# B&R Automation Studio project CarWashSimu (part 2)

#### Main.st - Init, cyclic, exit code
```iecst
PROGRAM _INIT
	(* Insert code here *)

END_PROGRAM

PROGRAM _CYCLIC
	(* Insert code here *)
	HPAlarm;
	CASE sHPolishState OF
		enWAIT:
			IF iHPolish.Cmd.Start = TRUE THEN
				sHPolishState				:= enSTART;
			END_IF;
		enSTART:
			IF (iHPolish.IO.diSensHPolish1 = FALSE) AND (iHPolish.IO.diSensHPolish2 = FALSE) AND (iHPolish.IO.diSensHPolish3 = FALSE) AND (iHPolish.IO.diSensHPolish4 = FALSE) THEN
				iHPolish.IO.doRelayLower	:= TRUE;
				iHPolish.IO.doRelayLift		:= FALSE;
			END_IF;
			IF (iHPolish.IO.diSensHPolish1 = TRUE) AND (iHPolish.IO.diSensHPolish2 = FALSE) AND (iHPolish.IO.diSensHPolish3 = FALSE) AND (iHPolish.IO.diSensHPolish4 = FALSE) THEN
				iHPolish.IO.doRelayLower	:= FALSE;
				iHPolish.IO.doRelayLift		:= FALSE;
				iHPolish.IO.doRelayBrush	:= TRUE;
				sHPolishState				:= enOPERATION;
			END_IF;
		enOPERATION:
			IF (iHPolish.IO.diSensHPolish1 = TRUE) AND (iHPolish.IO.diSensHPolish2 = FALSE) AND (iHPolish.IO.diSensHPolish3 = FALSE) AND (iHPolish.IO.diSensHPolish4 = FALSE) THEN
				iHPolish.IO.doRelayLower	:= FALSE;
				iHPolish.IO.doRelayLift	:= FALSE;
			END_IF;
			IF (iHPolish.IO.diSensHPolish1 = TRUE) AND (iHPolish.IO.diSensHPolish2 = TRUE) AND (iHPolish.IO.diSensHPolish3 = TRUE) AND (iHPolish.IO.diSensHPolish4 = FALSE) THEN
				iHPolish.IO.doRelayLower	:= FALSE;
				iHPolish.IO.doRelayLift	:= TRUE;
			END_IF;
			IF (iHPolish.IO.diSensHPolish1 = TRUE) AND (iHPolish.IO.diSensHPolish2 = TRUE) AND (iHPolish.IO.diSensHPolish3 = FALSE) AND (iHPolish.IO.diSensHPolish4 = FALSE) THEN
				iHPolish.IO.doRelayLower	:= FALSE;
				iHPolish.IO.doRelayLift	:= TRUE;
			END_IF;
			IF (iHPolish.IO.diSensHPolish1 = FALSE) AND (iHPolish.IO.diSensHPolish2 = FALSE) AND (iHPolish.IO.diSensHPolish3 = TRUE) AND (iHPolish.IO.diSensHPolish4 = FALSE) THEN
				iHPolish.IO.doRelayLower	:= TRUE;
				iHPolish.IO.doRelayLift	:= FALSE;
			END_IF;
			IF (iHPolish.IO.diSensHPolish1 = FALSE) AND (iHPolish.IO.diSensHPolish2 = FALSE) AND (iHPolish.IO.diSensHPolish3 = TRUE) AND (iHPolish.IO.diSensHPolish4 = TRUE) THEN
				iHPolish.IO.doRelayLower	:= FALSE;
				iHPolish.IO.doRelayLift	:= FALSE;
			END_IF;
			IF (iHPolish.IO.diSensHPolish1 = FALSE) AND (iHPolish.IO.diSensHPolish2 = FALSE) AND (iHPolish.IO.diSensHPolish3 = FALSE) AND (iHPolish.IO.diSensHPolish4 = FALSE) THEN
				iHPolish.IO.doRelayLower	:= FALSE;
				iHPolish.IO.doRelayLift	:= FALSE;
				iHPolish.IO.doRelayBrush	:= FALSE;
				iHPolish.Cmd.Start			:= FALSE;
				sHPolishState				:= enWAIT;
			END_IF;

		enERROR:
			iHPolish.IO.doRelayLower	:= FALSE;
			iHPolish.IO.doRelayLift		:= FALSE;
			iHPolish.IO.doRelayBrush	:= FALSE;
			iHPolish.Cmd.Start			:= FALSE;
			IF iHPolish.Cmd.ErrorReset=TRUE THEN
				iHPolish.Cmd.EStop:=FALSE;
				iHPolish.Cmd.ErrorReset:=FALSE;
				iHPolish.Status.Error:=FALSE;
				sHPolishState:=enSTART;
			END_IF;

	END_CASE;
END_PROGRAM

PROGRAM _EXIT
	(* Insert code here *)

END_PROGRAM
```

#### Types.typ - Local data types
```iecst
TYPE
	HorizontalPolishState_enum :
		(
		enWAIT,
		enSTART,
		enOPERATION,
		enERROR
		);
END_TYPE
```

#### Variables.var - Local variables
```iecst
VAR
	iHPolish : PolishCtrl_typ;
	sHPolishState : HorizontalPolishState_enum;
END_VAR
```

#### HPAlarm.st
```iecst
ACTION HPAlarm:
	IF iHPolish.Cmd.EStop=TRUE THEN
		MpAlarmXSet(gAlarmXCore,'EStopHPol');
		IF MpAlarmXCheckReaction(gAlarmXCore, 'EStopErr') THEN
			iHPolish.Status.Error:= TRUE ;
		END_IF
	ELSE
		MpAlarmXReset(gAlarmXCore,'EStopHPol');
	END_IF;
END_ACTION
```

### Types.typ
```iecst
TYPE
	PolishCmd_typ : 	STRUCT
		Start : BOOL;
		EStop : BOOL;
		Stop : BOOL;
		ErrorReset : USINT;
	END_STRUCT;
	PolishCtrl_typ : 	STRUCT
		Cmd : PolishCmd_typ;
		IO : PolishIOs_typ;
		Par : PolishParam_typ;
		Status : PolishStatus_typ;
	END_STRUCT;
	PolishIOs_typ : 	STRUCT
		doRelayLower : BOOL;
		doRelayBrush : BOOL;
		doRelayLift : BOOL;
		diSensHPolish2 : BOOL;
		diSensHPolish3 : BOOL;
		diSensHPolish4 : BOOL;
		diSensHPolish1 : BOOL;
	END_STRUCT;
	PolishParam_typ : 	STRUCT
		New_Member : BOOL;
	END_STRUCT;
	PolishStatus_typ : 	STRUCT
		Running : BOOL;
		Error : BOOL;
	END_STRUCT;
END_TYPE
```

### Program Logical/Source/Dist (IEC)

#### Types.typ
```iecst
TYPE
	DistanceState_enum :
		(
		enSTART,
		enDISTMOVE
		);
END_TYPE
```

#### Variables.var
```iecst
VAR
	a : REAL;
	Status1 : UINT;
	AuxAddress : UDINT;
	SizeAux : UDINT;
	pDistAux : REFERENCE TO Auxillary_typ;
	Status2 : UINT;
	EntryAddress : UDINT;
	SizeEntry : UDINT;
	pDistEntry : REFERENCE TO EntryCtrl_typ;
	sDistState : DistanceState_enum;
END_VAR
```

#### Main.st
```iecst
PROGRAM _INIT
	(* Insert code here *)
	Status1 := PV_xgetadr(ADR('Auxillary:iAuxillary'),ADR(AuxAddress),ADR(SizeAux));
	Status2 := PV_xgetadr(ADR('EntryCtrl:iEntry'),ADR(EntryAddress),ADR(SizeEntry));

END_PROGRAM

PROGRAM _CYCLIC
	(* Insert code here *)

	pDistAux	ACCESS AuxAddress;
	pDistEntry	ACCESS EntryAddress;

	CASE sDistState OF
		enSTART:
			IF pDistEntry.IO.diSensEntry = TRUE THEN
				sDistState		:= enDISTMOVE;
			END_IF;
		enDISTMOVE:
			IF pDistAux.doRelayConv = TRUE THEN
				iVa_Distance	:= iVa_Distance + 0.044;
			END_IF;
	END_CASE;

END_PROGRAM

PROGRAM _EXIT
	(* Insert code here *)

END_PROGRAM
```

### Program Logical/Source/HOpthpolish/HPolish

#### Main.st
```iecst
PROGRAM _INIT
	(* Insert code here *)

END_PROGRAM

PROGRAM _CYCLIC
	(* Insert code here *)

	CASE sHPolishState OF
		enWAIT:
			IF iHPolish.Cmd.Start = TRUE THEN
				sHPolishState				:= enSTART;
			END_IF;
		enSTART:
			IF (iHPolish.IO.diSensHPolish1 = FALSE) AND (iHPolish.IO.diSensHPolish2 = FALSE) AND (iHPolish.IO.diSensHPolish3 = FALSE) AND (iHPolish.IO.diSensHPolish4 = FALSE) THEN
				iHPolish.IO.doRelayLower	:= TRUE;
				iHPolish.IO.doRelayLift		:= FALSE;
			END_IF;
			IF (iHPolish.IO.diSensHPolish1 = TRUE) AND (iHPolish.IO.diSensHPolish2 = FALSE) AND (iHPolish.IO.diSensHPolish3 = FALSE) AND (iHPolish.IO.diSensHPolish4 = FALSE) THEN
				iHPolish.IO.doRelayLower	:= FALSE;
				iHPolish.IO.doRelayLift		:= FALSE;
				iHPolish.IO.doRelayBrush	:= TRUE;
				sHPolishState				:= enOPERATION;
			END_IF;
		enOPERATION:
			IF (iHPolish.IO.diSensHPolish1 = TRUE) AND (iHPolish.IO.diSensHPolish2 = FALSE) AND (iHPolish.IO.diSensHPolish3 = FALSE) AND (iHPolish.IO.diSensHPolish4 = FALSE) THEN
				iHPolish.IO.doRelayLower	:= FALSE;
				iHPolish.IO.doRelayLift	:= FALSE;
			END_IF;
			IF (iHPolish.IO.diSensHPolish1 = TRUE) AND (iHPolish.IO.diSensHPolish2 = TRUE) AND (iHPolish.IO.diSensHPolish3 = TRUE) AND (iHPolish.IO.diSensHPolish4 = FALSE) THEN
				iHPolish.IO.doRelayLower	:= FALSE;
				iHPolish.IO.doRelayLift	:= TRUE;
			END_IF;
			IF (iHPolish.IO.diSensHPolish1 = TRUE) AND (iHPolish.IO.diSensHPolish2 = TRUE) AND (iHPolish.IO.diSensHPolish3 = FALSE) AND (iHPolish.IO.diSensHPolish4 = FALSE) THEN
				iHPolish.IO.doRelayLower	:= FALSE;
				iHPolish.IO.doRelayLift	:= TRUE;
			END_IF;
			IF (iHPolish.IO.diSensHPolish1 = FALSE) AND (iHPolish.IO.diSensHPolish2 = FALSE) AND (iHPolish.IO.diSensHPolish3 = TRUE) AND (iHPolish.IO.diSensHPolish4 = FALSE) THEN
				iHPolish.IO.doRelayLower	:= TRUE;
				iHPolish.IO.doRelayLift	:= FALSE;
			END_IF;
			IF (iHPolish.IO.diSensHPolish1 = FALSE) AND (iHPolish.IO.diSensHPolish2 = FALSE) AND (iHPolish.IO.diSensHPolish3 = TRUE) AND (iHPolish.IO.diSensHPolish4 = TRUE) THEN
				iHPolish.IO.doRelayLower	:= FALSE;
				iHPolish.IO.doRelayLift	:= FALSE;
			END_IF;
			IF (iHPolish.IO.diSensHPolish1 = FALSE) AND (iHPolish.IO.diSensHPolish2 = FALSE) AND (iHPolish.IO.diSensHPolish3 = FALSE) AND (iHPolish.IO.diSensHPolish4 = FALSE) THEN
				iHPolish.IO.doRelayLower	:= FALSE;
				iHPolish.IO.doRelayLift	:= FALSE;
				iHPolish.IO.doRelayBrush	:= FALSE;
				iHPolish.Cmd.Start			:= FALSE;
				sHPolishState				:= enWAIT;
			END_IF;
	END_CASE;
END_PROGRAM

PROGRAM _EXIT
	(* Insert code here *)

END_PROGRAM
```

### HPolishCtrl.typ
```iecst
TYPE
	PolishCmd_typ : 	STRUCT
		Start : BOOL;
		EStop : BOOL;
		Stop : BOOL;
	END_STRUCT;
	PolishCtrl_typ : 	STRUCT
		Cmd : PolishCmd_typ;
		IO : PolishIOs_typ;
		Par : PolishParam_typ;
		Status : PolishStatus_typ;
	END_STRUCT;
	PolishIOs_typ : 	STRUCT
		doRelayLower : BOOL;
		doRelayBrush : BOOL;
		doRelayLift : BOOL;
		diSensHPolish2 : BOOL;
		diSensHPolish3 : BOOL;
		diSensHPolish4 : BOOL;
		diSensHPolish1 : BOOL;
	END_STRUCT;
	PolishParam_typ : 	STRUCT
<<<<<<< HEAD:Logical/Source/Optpolish/HPolishCtrl.typ
		New_Member : USINT;
=======
		New_Member : BOOL;
>>>>>>> edcf355ccd2dc5a058ed4214cc82538d90d7c920:Logical/Source/HOpthpolish/HPolishCtrl.typ
	END_STRUCT;
	PolishStatus_typ : 	STRUCT
		Running : BOOL;
		Error : BOOL;
	END_STRUCT;
END_TYPE
```

### Program Logical/Source/Optpolish/HPolishCtrl

#### Variables.var
```iecst
VAR
	iHPolish : PolishCtrl_typ;
END_VAR
```

#### Main.st
```iecst
PROGRAM _INIT
	(* Insert code here *)

END_PROGRAM

PROGRAM _CYCLIC
<<<<<<<< HEAD:Logical/Source/Optpolish/HPolishCtrl/Main.st
iHPolish;
========
	(* Insert code here *)

	a	:= a + 0.44;

>>>>>>>> edcf355ccd2dc5a058ed4214cc82538d90d7c920:Logical/Dist/Main.st
END_PROGRAM

PROGRAM _EXIT
	(* Insert code here *)

END_PROGRAM
```

- Visualisation Logical/mappView (not shown)

### Program Logical/Dist

#### Variables.var
```iecst
VAR
	a : REAL;
END_VAR
```

#### Main.st
```iecst
PROGRAM _INIT
	(* Insert code here *)

END_PROGRAM

PROGRAM _CYCLIC
	(* Insert code here *)

	a	:= a + 0.44;

END_PROGRAM

PROGRAM _EXIT
	(* Insert code here *)

END_PROGRAM
```

Listed in the project but not available here: Logical/Libraries/ComTCP/ComTCP_L/MNG_InternalTyp.hpp, Logical/Libraries/ComTCP/ComTCP_L/MNG_ComHdlr.hpp, Logical/Libraries/ComTCP/ComTCP_L/MNG_ComHdlr.cpp, Logical/Documentation, Logical/Source/VBrush/VBrushCtrl/Types.typ, Logical/Source/Drying/DryHCtrl/Types.typ, Logical/Source/Infrastructure/RecipeCtrl/RecipeCtrl, Logical/Source/Optpolish/HPolish
